(* Logix 5000 project; controller oki_4_19 vendor 1 type 14 code 77 rev 20.12; software revision 20.01 *)

TASK MainTask (continuous, watchdog 500 ms) : MainProgram

MODULES
   Controller : vendor 1 type 14 code 77 (CompactLogixL32EController 0, rev 20.12)
      LocalENB : 1769-L32E Ethernet Port (CompactLogixL32Ethernet 1, rev 20.11)
      Local : CompactBus (CompactVirtualAdapter 3, rev 20.11)
         DC_INPUT_1 : 1769-IQ16 (Compact 1, rev 1.1, Input RPI 20 ms)
         DC_OUTPUT_1 : 1769-OB16 (Compact 2, rev 2.1, Output RPI 20 ms)
END_MODULES

VAR_GLOBAL   (* controller tags *)
   LED : ALIAS FOR Local:2:O.Data.15;
   SW1 : ALIAS FOR Local:1:I.Data.1;
   SW2 : ALIAS FOR Local:1:I.Data.2;
   SW3 : ALIAS FOR Local:1:I.Data.3;
END_VAR

PROGRAM MainProgram   (* main routine MainRoutine *)

ROUTINE MainRoutine   (* ladder *)
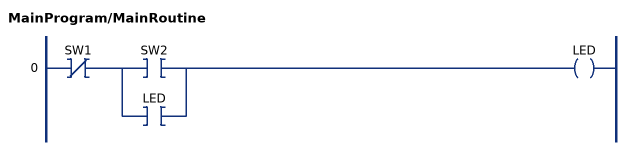
   0: XIO(SW1)[XIC(SW2) ,XIC(LED) ]OTE(LED);
END_ROUTINE
END_PROGRAM
